SYSTEM DRILL_MVCL (* Drill System Model+View+Control+HMI with shared simulation clock *)
  (* Standard: 61499-1; Classification: Simulation; ApplicationDomain: Transfer Lines; Function: Drilling *)
  (* Version 0.2, 2007-07-07, JHC, Holobloc Inc, Added MODEL.CLOCK.CLK_DLY. *)
  (* Version 0.1, 2006-03-06, JHC, Holobloc Inc, Modified for new MACH_CTL. *)
  (* Version 0.0, 2004-09-26, JHC, Rockwell Automation, Derived from DRILL_MVL. *)
  DEVICE MODEL : FRAME_DEVICE(BOUNDS := [475,100,190,360])
    RESOURCE CLOCK : EMB_RES
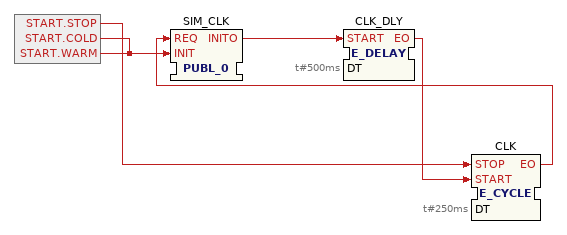
      FBS
        CLK : E_CYCLE(DT := t#250ms);
        SIM_CLK : PUBL_0;
        CLK_DLY : E_DELAY(DT := t#500ms); (* Wait for everything to initialize, then start simulation *)
      END_FBS
      EVENT_CONNECTIONS
        CLK.EO TO SIM_CLK.REQ;
        START.STOP TO CLK.STOP;
        START.COLD TO SIM_CLK.INIT;
        START.WARM TO SIM_CLK.INIT;
        SIM_CLK.INITO TO CLK_DLY.START;
        CLK_DLY.EO TO CLK.START;
      END_CONNECTIONS
    END_RESOURCE
    RESOURCE SUPPLY_MDL : EMB_RES
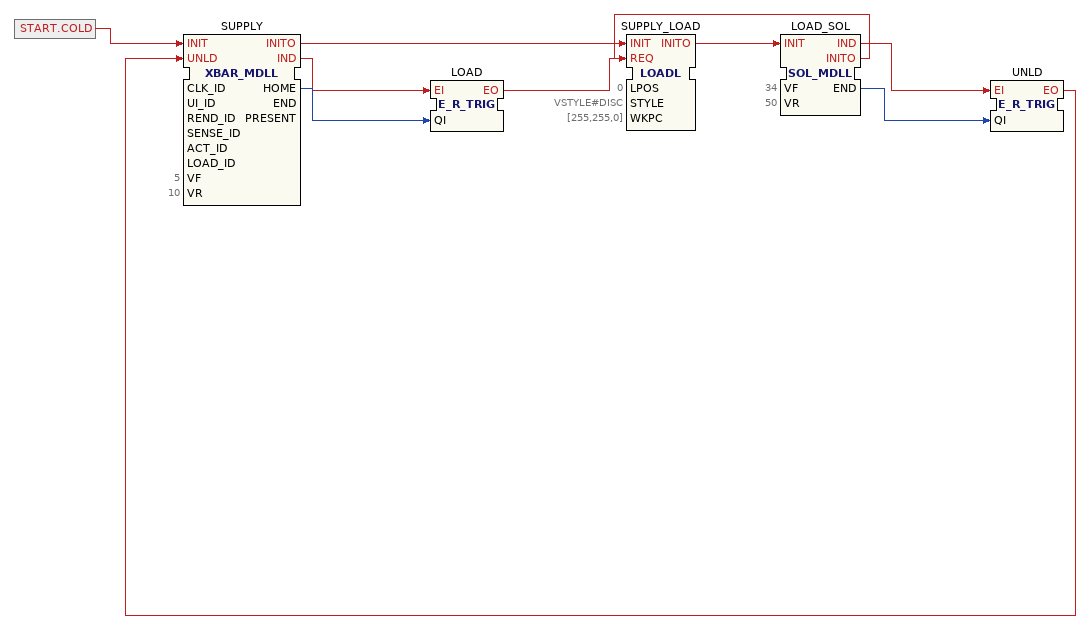
      FBS
        SUPPLY : XBAR_MDLL(VF := 5, VR := 10);
        LOAD_SOL : SOL_MDLL(VF := 34, VR := 50);
        UNLD : E_R_TRIG;
        LOAD : E_R_TRIG;
        SUPPLY_LOAD : LOADL(LPOS := 0, STYLE := VSTYLE#DISC, WKPC := [255,255,0]);
      END_FBS
      EVENT_CONNECTIONS
        START.COLD TO SUPPLY.INIT;
        LOAD_SOL.IND TO UNLD.EI;
        SUPPLY.IND TO LOAD.EI;
        UNLD.EO TO SUPPLY.UNLD;
        SUPPLY.INITO TO SUPPLY_LOAD.INIT;
        SUPPLY_LOAD.INITO TO LOAD_SOL.INIT;
        LOAD_SOL.INITO TO SUPPLY_LOAD.REQ;
        LOAD.EO TO SUPPLY_LOAD.REQ;
      END_CONNECTIONS
      DATA_CONNECTIONS
        LOAD_SOL.END TO UNLD.QI;
        SUPPLY.HOME TO LOAD.QI;
      END_CONNECTIONS
    END_RESOURCE
    RESOURCE SLIDE_MDL : EMB_RES
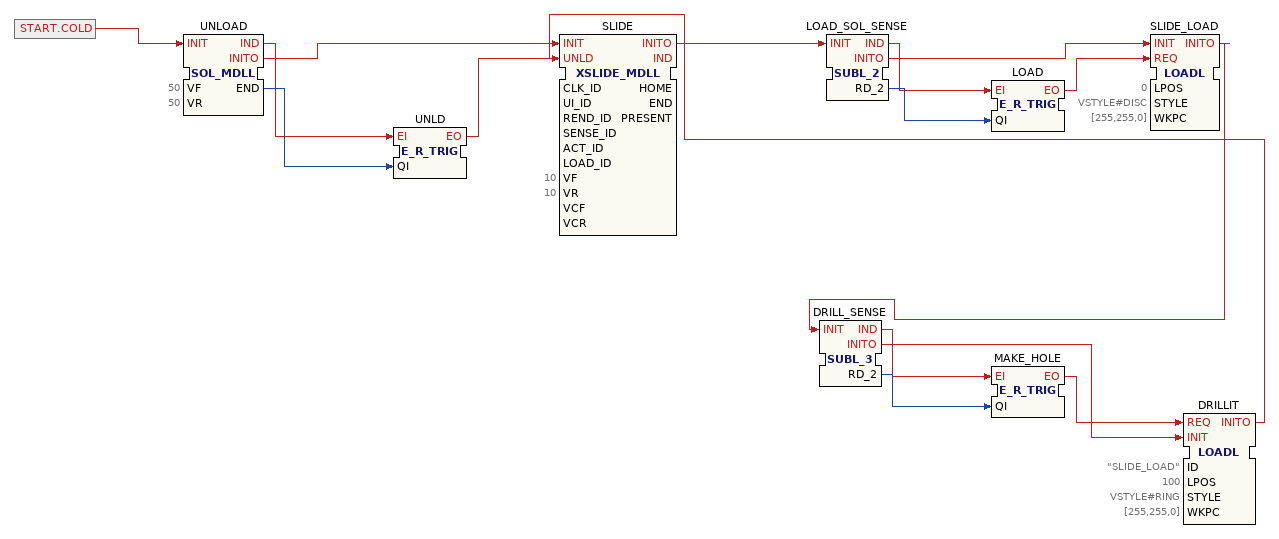
      FBS
        SLIDE : XSLIDE_MDLL(VF := 10, VR := 10);
        UNLOAD : SOL_MDLL(VF := 50, VR := 50);
        DRILL_SENSE : SUBL_3;
        MAKE_HOLE : E_R_TRIG;
        UNLD : E_R_TRIG;
        LOAD_SOL_SENSE : SUBL_2;
        LOAD : E_R_TRIG;
        SLIDE_LOAD : LOADL(LPOS := 0, STYLE := VSTYLE#DISC, WKPC := [255,255,0]);
        DRILLIT : LOADL(ID := "SLIDE_LOAD", LPOS := 100, STYLE := VSTYLE#RING, WKPC := [255,255,0]);
      END_FBS
      EVENT_CONNECTIONS
        DRILL_SENSE.IND TO MAKE_HOLE.EI;
        UNLOAD.IND TO UNLD.EI;
        UNLD.EO TO SLIDE.UNLD;
        LOAD_SOL_SENSE.IND TO LOAD.EI;
        START.COLD TO UNLOAD.INIT;
        UNLOAD.INITO TO SLIDE.INIT;
        SLIDE.INITO TO LOAD_SOL_SENSE.INIT;
        LOAD_SOL_SENSE.INITO TO SLIDE_LOAD.INIT;
        LOAD.EO TO SLIDE_LOAD.REQ;
        MAKE_HOLE.EO TO DRILLIT.REQ;
        DRILLIT.INITO TO SLIDE.UNLD;
        SLIDE_LOAD.INITO TO DRILL_SENSE.INIT;
        DRILL_SENSE.INITO TO DRILLIT.INIT;
      END_CONNECTIONS
      DATA_CONNECTIONS
        DRILL_SENSE.RD_2 TO MAKE_HOLE.QI;
        UNLOAD.END TO UNLD.QI;
        LOAD_SOL_SENSE.RD_2 TO LOAD.QI;
      END_CONNECTIONS
    END_RESOURCE
    RESOURCE DRILL_MDL : EMB_RES
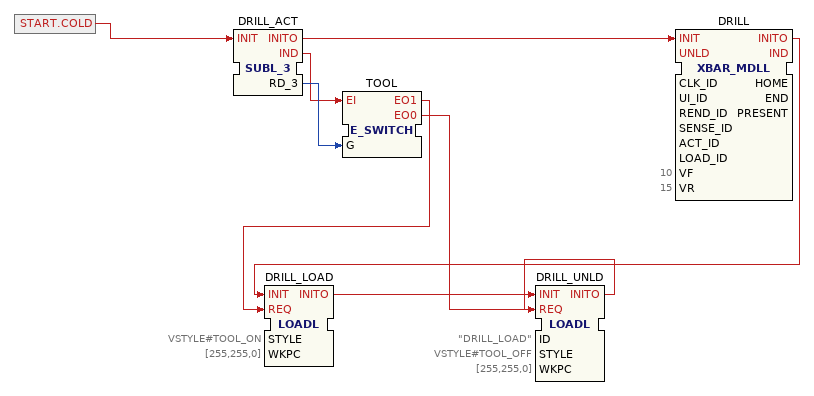
      FBS
        DRILL : XBAR_MDLL(VF := 10, VR := 15);
        DRILL_ACT : SUBL_3;
        TOOL : E_SWITCH;
        DRILL_LOAD : LOADL(STYLE := VSTYLE#TOOL_ON, WKPC := [255,255,0]);
        DRILL_UNLD : LOADL(ID := "DRILL_LOAD", STYLE := VSTYLE#TOOL_OFF, WKPC := [255,255,0]);
      END_FBS
      EVENT_CONNECTIONS
        START.COLD TO DRILL_ACT.INIT;
        DRILL_ACT.INITO TO DRILL.INIT;
        DRILL.INITO TO DRILL_LOAD.INIT;
        DRILL_LOAD.INITO TO DRILL_UNLD.INIT;
        DRILL_ACT.IND TO TOOL.EI;
        TOOL.EO1 TO DRILL_LOAD.REQ;
        TOOL.EO0 TO DRILL_UNLD.REQ;
        DRILL_UNLD.INITO TO DRILL_UNLD.REQ;
      END_CONNECTIONS
      DATA_CONNECTIONS
        DRILL_ACT.RD_3 TO TOOL.G;
      END_CONNECTIONS
    END_RESOURCE
    RESOURCE TAKEOFF_MDL : EMB_RES
      FBS
        UNLOAD_SENSE : SUBL_2;
        TAKEOFF : XBAR_MDLL(VF := 5, VR := 10);
        UNLD : E_R_TRIG;
        LOAD : E_R_TRIG;
        TAKEOFF_LOAD : LOADL(LPOS := 0, STYLE := VSTYLE#RING, WKPC := [255,255,0]);
      END_FBS
      EVENT_CONNECTIONS
        START.COLD TO UNLOAD_SENSE.INIT;
        UNLD.EO TO TAKEOFF.UNLD;
        TAKEOFF.IND TO UNLD.EI;
        TAKEOFF.INITO TO TAKEOFF.UNLD;
        UNLOAD_SENSE.IND TO LOAD.EI;
        UNLOAD_SENSE.INITO TO TAKEOFF_LOAD.INIT;
        TAKEOFF_LOAD.INITO TO TAKEOFF.INIT;
        LOAD.EO TO TAKEOFF_LOAD.REQ;
      END_CONNECTIONS
      DATA_CONNECTIONS
        TAKEOFF.END TO UNLD.QI;
        UNLOAD_SENSE.RD_2 TO LOAD.QI;
      END_CONNECTIONS
    END_RESOURCE
    RESOURCE INPUT_VIEW : VIEW_PANEL(DIA := 30, SIZE := [6,5], VERTICAL := 1)
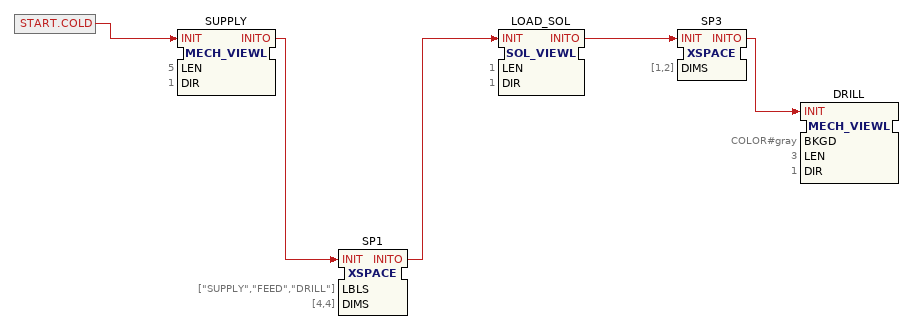
      FBS
        SUPPLY : MECH_VIEWL(LEN := 5, DIR := 1); (* Supply transfer mechanism *)
        SP1 : XSPACE(LBLS := ["SUPPLY","FEED","DRILL"], DIMS := [4,4]);
        LOAD_SOL : SOL_VIEWL(LEN := 1, DIR := 1); (* Loader mechanism *)
        SP3 : XSPACE(DIMS := [1,2]);
        DRILL : MECH_VIEWL(BKGD := COLOR#gray, LEN := 3, DIR := 1);
      END_FBS
      EVENT_CONNECTIONS
        START.COLD TO SUPPLY.INIT;
        SUPPLY.INITO TO SP1.INIT;
        SP1.INITO TO LOAD_SOL.INIT;
        LOAD_SOL.INITO TO SP3.INIT;
        SP3.INITO TO DRILL.INIT;
      END_CONNECTIONS
    END_RESOURCE
    RESOURCE OUTPUT_VIEW : VIEW_PANEL(DIA := 30, SIZE := [6,5])
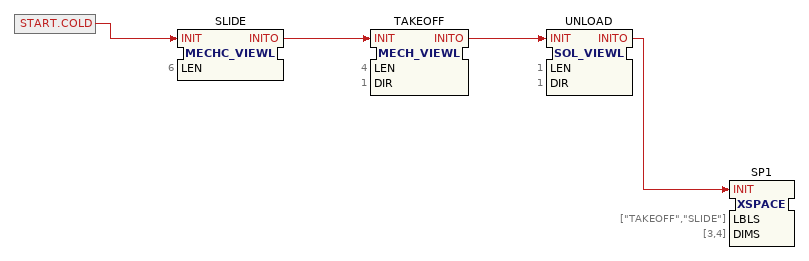
      FBS
        SLIDE : MECHC_VIEWL(LEN := 6);
        TAKEOFF : MECH_VIEWL(LEN := 4, DIR := 1); (* Takeoff Transfer *)
        UNLOAD : SOL_VIEWL(LEN := 1, DIR := 1); (* Unloader Mechanism *)
        SP1 : XSPACE(LBLS := ["TAKEOFF","SLIDE"], DIMS := [3,4]);
      END_FBS
      EVENT_CONNECTIONS
        START.COLD TO SLIDE.INIT;
        SLIDE.INITO TO TAKEOFF.INIT;
        TAKEOFF.INITO TO UNLOAD.INIT;
        UNLOAD.INITO TO SP1.INIT;
      END_CONNECTIONS
    END_RESOURCE
  END_DEVICE
  DEVICE CONTROL : FRAME_DEVICE(BOUNDS := [100,100,375,360], GRID := [6,2])
    RESOURCE SUPPLY_SENSORS : PANEL_RESOURCE
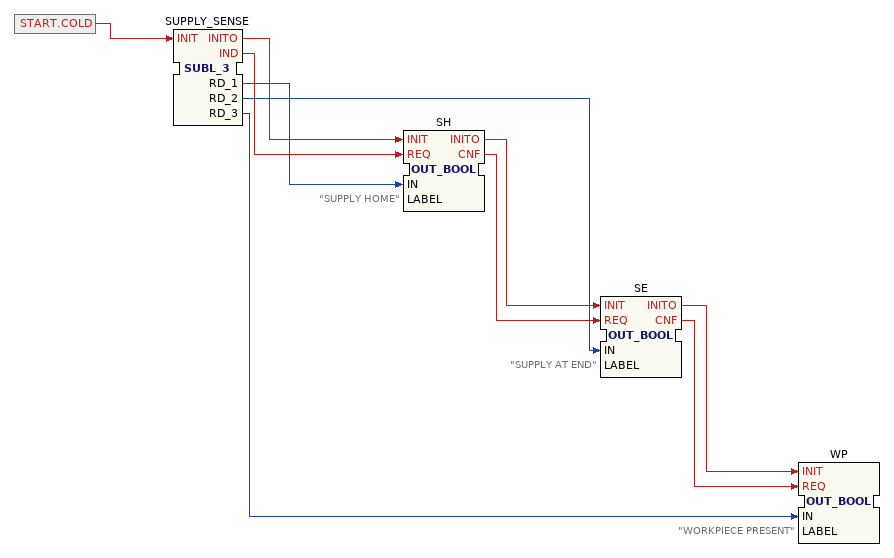
      FBS
        SUPPLY_SENSE : SUBL_3;
        SH : OUT_BOOL(LABEL := "SUPPLY HOME");
        SE : OUT_BOOL(LABEL := "SUPPLY AT END");
        WP : OUT_BOOL(LABEL := "WORKPIECE PRESENT");
      END_FBS
      EVENT_CONNECTIONS
        START.COLD TO SUPPLY_SENSE.INIT;
        SUPPLY_SENSE.INITO TO SH.INIT;
        SH.INITO TO SE.INIT;
        SE.INITO TO WP.INIT;
        SUPPLY_SENSE.IND TO SH.REQ;
        SH.CNF TO SE.REQ;
        SE.CNF TO WP.REQ;
      END_CONNECTIONS
      DATA_CONNECTIONS
        SUPPLY_SENSE.RD_1 TO SH.IN;
        SUPPLY_SENSE.RD_2 TO SE.IN;
        SUPPLY_SENSE.RD_3 TO WP.IN;
      END_CONNECTIONS
    END_RESOURCE
    RESOURCE SUPPLY_ACTUATORS : PANEL_RESOURCE(ROWS := 3)
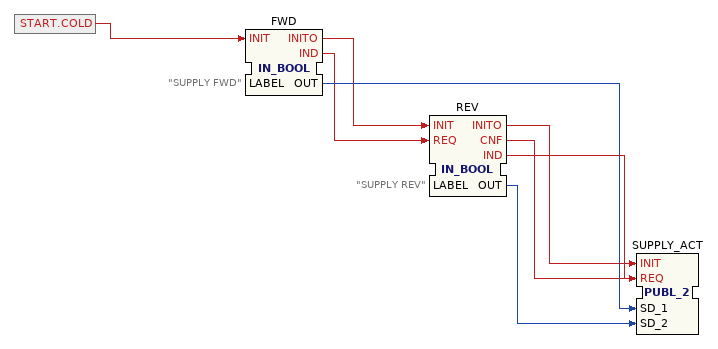
      FBS
        FWD : IN_BOOL(LABEL := "SUPPLY FWD");
        REV : IN_BOOL(LABEL := "SUPPLY REV");
        SUPPLY_ACT : PUBL_2;
      END_FBS
      EVENT_CONNECTIONS
        START.COLD TO FWD.INIT;
        FWD.INITO TO REV.INIT;
        REV.INITO TO SUPPLY_ACT.INIT;
        FWD.IND TO REV.REQ;
        REV.CNF TO SUPPLY_ACT.REQ;
        REV.IND TO SUPPLY_ACT.REQ;
      END_CONNECTIONS
      DATA_CONNECTIONS
        FWD.OUT TO SUPPLY_ACT.SD_1;
        REV.OUT TO SUPPLY_ACT.SD_2;
      END_CONNECTIONS
    END_RESOURCE
    RESOURCE LOAD_SENSORS : PANEL_RESOURCE
      FBS
        LOAD_SOL_SENSE : SUBL_2;
        HOME : OUT_BOOL(LABEL := "LOADER HOME");
        END : OUT_BOOL(LABEL := "LOADER AT END");
      END_FBS
      EVENT_CONNECTIONS
        START.COLD TO LOAD_SOL_SENSE.INIT;
        LOAD_SOL_SENSE.INITO TO HOME.INIT;
        HOME.INITO TO END.INIT;
        LOAD_SOL_SENSE.IND TO HOME.REQ;
        HOME.CNF TO END.REQ;
      END_CONNECTIONS
      DATA_CONNECTIONS
        LOAD_SOL_SENSE.RD_1 TO HOME.IN;
        LOAD_SOL_SENSE.RD_2 TO END.IN;
      END_CONNECTIONS
    END_RESOURCE
    RESOURCE LOAD_ACTUATORS : PANEL_RESOURCE(ROWS := 3)
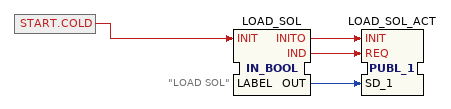
      FBS
        LOAD_SOL : IN_BOOL(LABEL := "LOAD SOL");
        LOAD_SOL_ACT : PUBL_1;
      END_FBS
      EVENT_CONNECTIONS
        START.COLD TO LOAD_SOL.INIT;
        LOAD_SOL.INITO TO LOAD_SOL_ACT.INIT;
        LOAD_SOL.IND TO LOAD_SOL_ACT.REQ;
      END_CONNECTIONS
      DATA_CONNECTIONS
        LOAD_SOL.OUT TO LOAD_SOL_ACT.SD_1;
      END_CONNECTIONS
    END_RESOURCE
    RESOURCE SLIDE_SENSORS : PANEL_RESOURCE
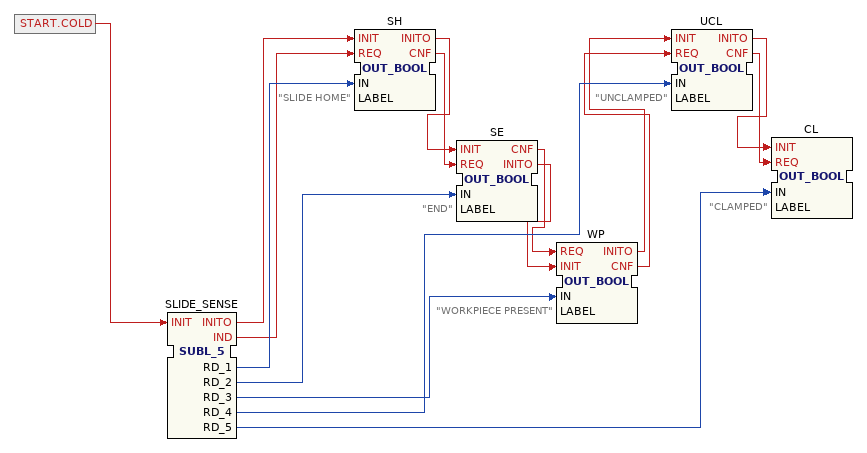
      FBS
        SLIDE_SENSE : SUBL_5;
        SH : OUT_BOOL(LABEL := "SLIDE HOME");
        SE : OUT_BOOL(LABEL := "END");
        UCL : OUT_BOOL(LABEL := "UNCLAMPED");
        CL : OUT_BOOL(LABEL := "CLAMPED");
        WP : OUT_BOOL(LABEL := "WORKPIECE PRESENT");
      END_FBS
      EVENT_CONNECTIONS
        START.COLD TO SLIDE_SENSE.INIT;
        SLIDE_SENSE.INITO TO SH.INIT;
        SH.INITO TO SE.INIT;
        UCL.INITO TO CL.INIT;
        SLIDE_SENSE.IND TO SH.REQ;
        SH.CNF TO SE.REQ;
        UCL.CNF TO CL.REQ;
        SE.CNF TO WP.REQ;
        SE.INITO TO WP.INIT;
        WP.INITO TO UCL.INIT;
        WP.CNF TO UCL.REQ;
      END_CONNECTIONS
      DATA_CONNECTIONS
        SLIDE_SENSE.RD_1 TO SH.IN;
        SLIDE_SENSE.RD_2 TO SE.IN;
        SLIDE_SENSE.RD_3 TO WP.IN;
        SLIDE_SENSE.RD_4 TO UCL.IN;
        SLIDE_SENSE.RD_5 TO CL.IN;
      END_CONNECTIONS
    END_RESOURCE
    RESOURCE SLIDE_ACTUATORS : PANEL_RESOURCE(ROWS := 3)
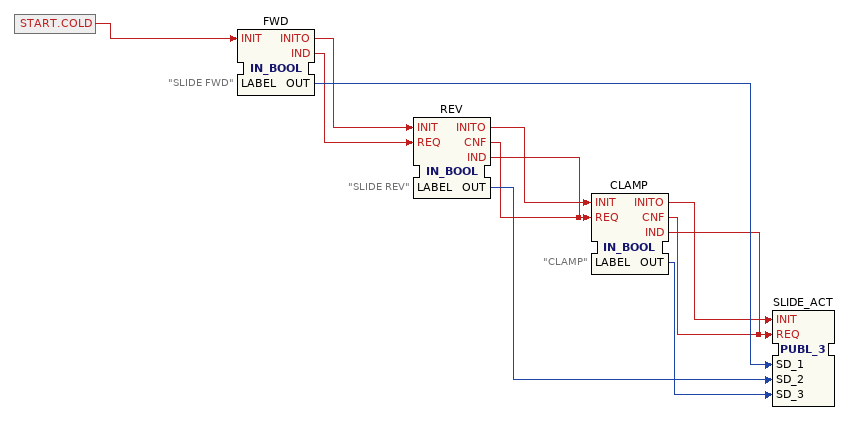
      FBS
        FWD : IN_BOOL(LABEL := "SLIDE FWD");
        REV : IN_BOOL(LABEL := "SLIDE REV");
        CLAMP : IN_BOOL(LABEL := "CLAMP");
        SLIDE_ACT : PUBL_3;
      END_FBS
      EVENT_CONNECTIONS
        START.COLD TO FWD.INIT;
        FWD.INITO TO REV.INIT;
        REV.INITO TO CLAMP.INIT;
        CLAMP.INITO TO SLIDE_ACT.INIT;
        FWD.IND TO REV.REQ;
        REV.CNF TO CLAMP.REQ;
        REV.IND TO CLAMP.REQ;
        CLAMP.CNF TO SLIDE_ACT.REQ;
        CLAMP.IND TO SLIDE_ACT.REQ;
      END_CONNECTIONS
      DATA_CONNECTIONS
        FWD.OUT TO SLIDE_ACT.SD_1;
        REV.OUT TO SLIDE_ACT.SD_2;
        CLAMP.OUT TO SLIDE_ACT.SD_3;
      END_CONNECTIONS
    END_RESOURCE
    RESOURCE DRILL_SENSORS : PANEL_RESOURCE
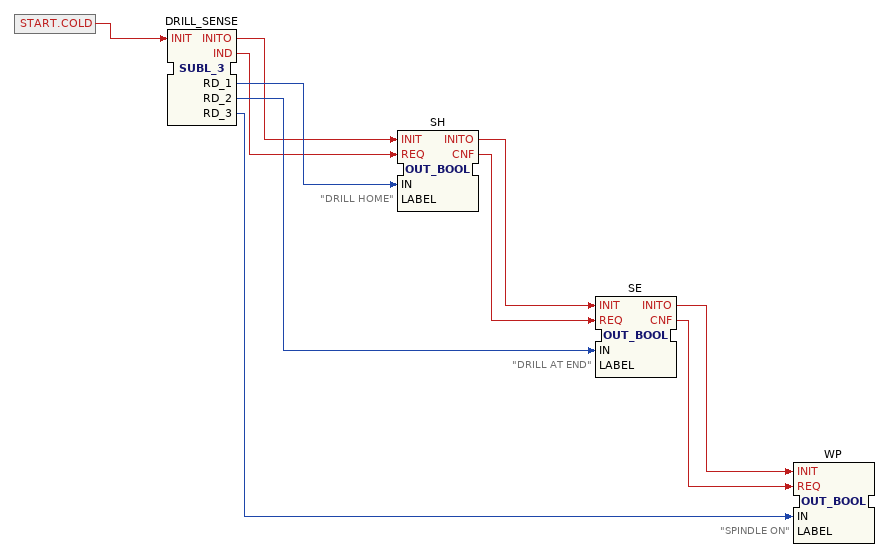
      FBS
        DRILL_SENSE : SUBL_3;
        SH : OUT_BOOL(LABEL := "DRILL HOME");
        SE : OUT_BOOL(LABEL := "DRILL AT END");
        WP : OUT_BOOL(LABEL := "SPINDLE ON");
      END_FBS
      EVENT_CONNECTIONS
        START.COLD TO DRILL_SENSE.INIT;
        DRILL_SENSE.INITO TO SH.INIT;
        SH.INITO TO SE.INIT;
        SE.INITO TO WP.INIT;
        DRILL_SENSE.IND TO SH.REQ;
        SH.CNF TO SE.REQ;
        SE.CNF TO WP.REQ;
      END_CONNECTIONS
      DATA_CONNECTIONS
        DRILL_SENSE.RD_1 TO SH.IN;
        DRILL_SENSE.RD_2 TO SE.IN;
        DRILL_SENSE.RD_3 TO WP.IN;
      END_CONNECTIONS
    END_RESOURCE
    RESOURCE DRILL_ACTUATORS : PANEL_RESOURCE(ROWS := 3)
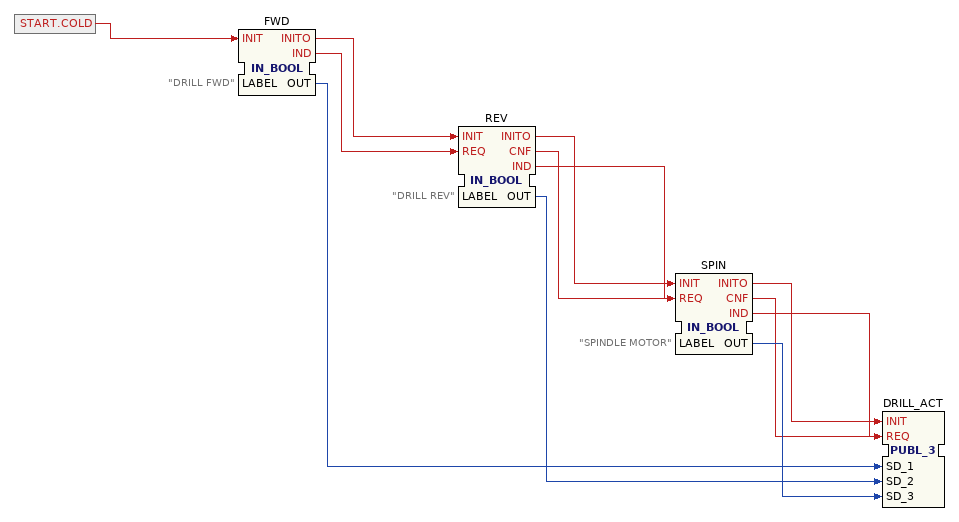
      FBS
        FWD : IN_BOOL(LABEL := "DRILL FWD");
        REV : IN_BOOL(LABEL := "DRILL REV");
        SPIN : IN_BOOL(LABEL := "SPINDLE MOTOR");
        DRILL_ACT : PUBL_3;
      END_FBS
      EVENT_CONNECTIONS
        START.COLD TO FWD.INIT;
        FWD.INITO TO REV.INIT;
        REV.INITO TO SPIN.INIT;
        SPIN.INITO TO DRILL_ACT.INIT;
        FWD.IND TO REV.REQ;
        REV.CNF TO SPIN.REQ;
        REV.IND TO SPIN.REQ;
        SPIN.CNF TO DRILL_ACT.REQ;
        SPIN.IND TO DRILL_ACT.REQ;
      END_CONNECTIONS
      DATA_CONNECTIONS
        FWD.OUT TO DRILL_ACT.SD_1;
        REV.OUT TO DRILL_ACT.SD_2;
        SPIN.OUT TO DRILL_ACT.SD_3;
      END_CONNECTIONS
    END_RESOURCE
    RESOURCE UNLOAD_SENSORS : PANEL_RESOURCE
      FBS
        UNLOAD_SENSE : SUBL_2;
        HOME : OUT_BOOL(LABEL := "UNLOADER HOME");
        END : OUT_BOOL(LABEL := "UNLOADER AT END");
      END_FBS
      EVENT_CONNECTIONS
        START.COLD TO UNLOAD_SENSE.INIT;
        UNLOAD_SENSE.INITO TO HOME.INIT;
        HOME.INITO TO END.INIT;
        UNLOAD_SENSE.IND TO HOME.REQ;
        HOME.CNF TO END.REQ;
      END_CONNECTIONS
      DATA_CONNECTIONS
        UNLOAD_SENSE.RD_1 TO HOME.IN;
        UNLOAD_SENSE.RD_2 TO END.IN;
      END_CONNECTIONS
    END_RESOURCE
    RESOURCE UNLOAD_ACTUATORS : PANEL_RESOURCE(ROWS := 3)
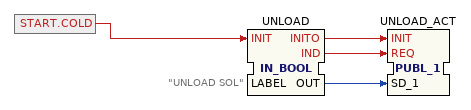
      FBS
        UNLOAD : IN_BOOL(LABEL := "UNLOAD SOL");
        UNLOAD_ACT : PUBL_1;
      END_FBS
      EVENT_CONNECTIONS
        START.COLD TO UNLOAD.INIT;
        UNLOAD.INITO TO UNLOAD_ACT.INIT;
        UNLOAD.IND TO UNLOAD_ACT.REQ;
      END_CONNECTIONS
      DATA_CONNECTIONS
        UNLOAD.OUT TO UNLOAD_ACT.SD_1;
      END_CONNECTIONS
    END_RESOURCE
    RESOURCE TAKEOFF_SENSORS : PANEL_RESOURCE
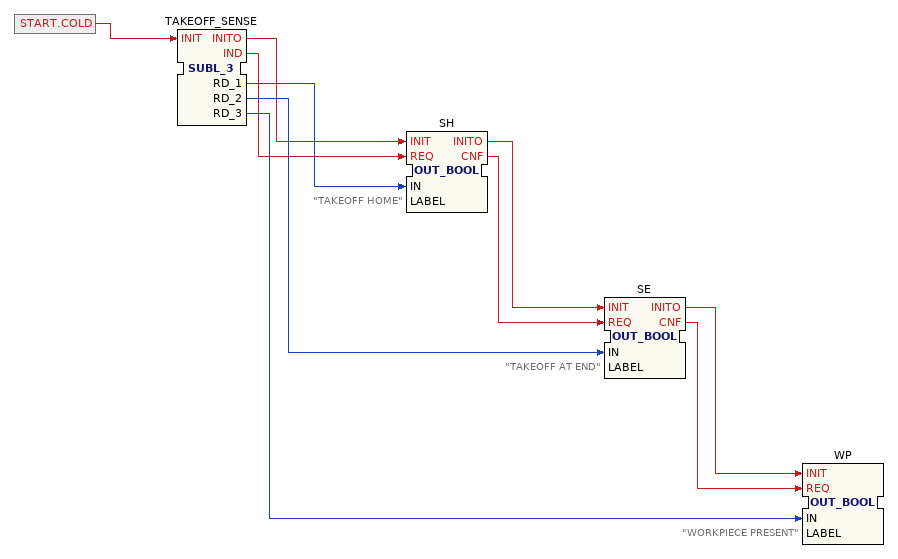
      FBS
        TAKEOFF_SENSE : SUBL_3;
        SH : OUT_BOOL(LABEL := "TAKEOFF HOME");
        SE : OUT_BOOL(LABEL := "TAKEOFF AT END");
        WP : OUT_BOOL(LABEL := "WORKPIECE PRESENT");
      END_FBS
      EVENT_CONNECTIONS
        START.COLD TO TAKEOFF_SENSE.INIT;
        TAKEOFF_SENSE.INITO TO SH.INIT;
        SH.INITO TO SE.INIT;
        SE.INITO TO WP.INIT;
        TAKEOFF_SENSE.IND TO SH.REQ;
        SH.CNF TO SE.REQ;
        SE.CNF TO WP.REQ;
      END_CONNECTIONS
      DATA_CONNECTIONS
        TAKEOFF_SENSE.RD_1 TO SH.IN;
        TAKEOFF_SENSE.RD_2 TO SE.IN;
        TAKEOFF_SENSE.RD_3 TO WP.IN;
      END_CONNECTIONS
    END_RESOURCE
    RESOURCE TAKEOFF_ACTUATORS : PANEL_RESOURCE(ROWS := 3)
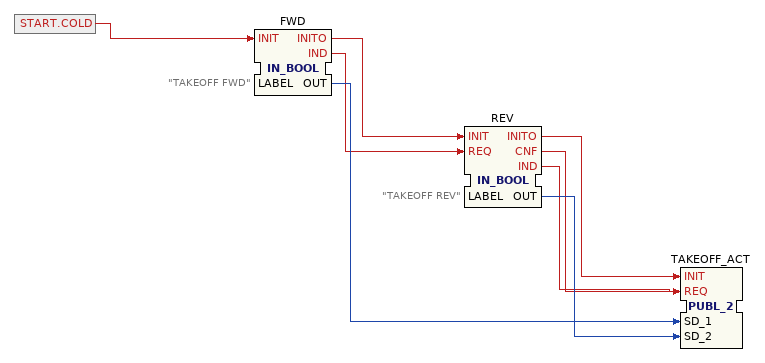
      FBS
        FWD : IN_BOOL(LABEL := "TAKEOFF FWD");
        REV : IN_BOOL(LABEL := "TAKEOFF REV");
        TAKEOFF_ACT : PUBL_2;
      END_FBS
      EVENT_CONNECTIONS
        START.COLD TO FWD.INIT;
        FWD.INITO TO REV.INIT;
        REV.INITO TO TAKEOFF_ACT.INIT;
        FWD.IND TO REV.REQ;
        REV.CNF TO TAKEOFF_ACT.REQ;
        REV.IND TO TAKEOFF_ACT.REQ;
      END_CONNECTIONS
      DATA_CONNECTIONS
        FWD.OUT TO TAKEOFF_ACT.SD_1;
        REV.OUT TO TAKEOFF_ACT.SD_2;
      END_CONNECTIONS
    END_RESOURCE
    RESOURCE SUPPLY : EMB_RES
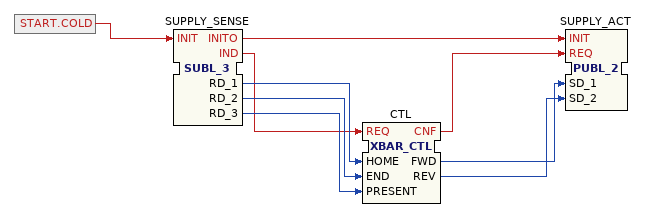
      FBS
        SUPPLY_SENSE : SUBL_3;
        CTL : XBAR_CTL;
        SUPPLY_ACT : PUBL_2;
      END_FBS
      EVENT_CONNECTIONS
        START.COLD TO SUPPLY_SENSE.INIT;
        SUPPLY_SENSE.INITO TO SUPPLY_ACT.INIT;
        SUPPLY_SENSE.IND TO CTL.REQ;
        CTL.CNF TO SUPPLY_ACT.REQ;
      END_CONNECTIONS
      DATA_CONNECTIONS
        SUPPLY_SENSE.RD_1 TO CTL.HOME;
        SUPPLY_SENSE.RD_2 TO CTL.END;
        SUPPLY_SENSE.RD_3 TO CTL.PRESENT;
        CTL.FWD TO SUPPLY_ACT.SD_1;
        CTL.REV TO SUPPLY_ACT.SD_2;
      END_CONNECTIONS
    END_RESOURCE
    RESOURCE LOAD : EMB_RES
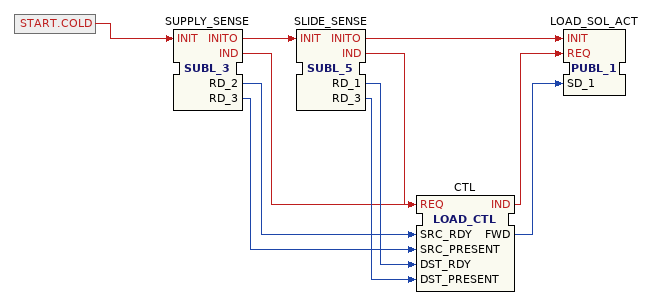
      FBS
        SUPPLY_SENSE : SUBL_3;
        SLIDE_SENSE : SUBL_5;
        CTL : LOAD_CTL;
        LOAD_SOL_ACT : PUBL_1;
      END_FBS
      EVENT_CONNECTIONS
        START.COLD TO SUPPLY_SENSE.INIT;
        SUPPLY_SENSE.INITO TO SLIDE_SENSE.INIT;
        SLIDE_SENSE.INITO TO LOAD_SOL_ACT.INIT;
        SUPPLY_SENSE.IND TO CTL.REQ;
        SLIDE_SENSE.IND TO CTL.REQ;
        CTL.IND TO LOAD_SOL_ACT.REQ;
      END_CONNECTIONS
      DATA_CONNECTIONS
        SUPPLY_SENSE.RD_2 TO CTL.SRC_RDY;
        SUPPLY_SENSE.RD_3 TO CTL.SRC_PRESENT;
        SLIDE_SENSE.RD_1 TO CTL.DST_RDY;
        CTL.FWD TO LOAD_SOL_ACT.SD_1;
        SLIDE_SENSE.RD_3 TO CTL.DST_PRESENT;
      END_CONNECTIONS
    END_RESOURCE
    RESOURCE SLIDE : EMB_RES
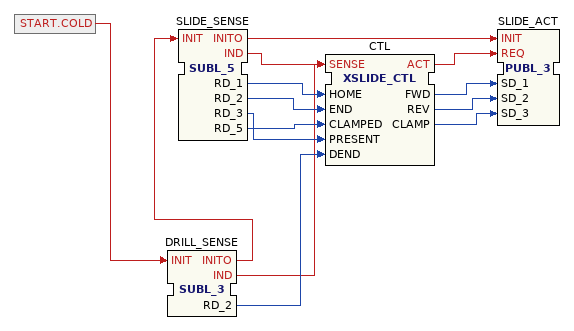
      FBS
        DRILL_SENSE : SUBL_3;
        SLIDE_SENSE : SUBL_5;
        CTL : XSLIDE_CTL;
        SLIDE_ACT : PUBL_3;
      END_FBS
      EVENT_CONNECTIONS
        START.COLD TO DRILL_SENSE.INIT;
        DRILL_SENSE.INITO TO SLIDE_SENSE.INIT;
        SLIDE_SENSE.INITO TO SLIDE_ACT.INIT;
        SLIDE_SENSE.IND TO CTL.SENSE;
        DRILL_SENSE.IND TO CTL.SENSE;
        CTL.ACT TO SLIDE_ACT.REQ;
      END_CONNECTIONS
      DATA_CONNECTIONS
        SLIDE_SENSE.RD_1 TO CTL.HOME;
        SLIDE_SENSE.RD_2 TO CTL.END;
        DRILL_SENSE.RD_2 TO CTL.DEND;
        CTL.FWD TO SLIDE_ACT.SD_1;
        CTL.REV TO SLIDE_ACT.SD_2;
        CTL.CLAMP TO SLIDE_ACT.SD_3;
        SLIDE_SENSE.RD_3 TO CTL.PRESENT;
        SLIDE_SENSE.RD_5 TO CTL.CLAMPED;
      END_CONNECTIONS
    END_RESOURCE
    RESOURCE DRILL : EMB_RES
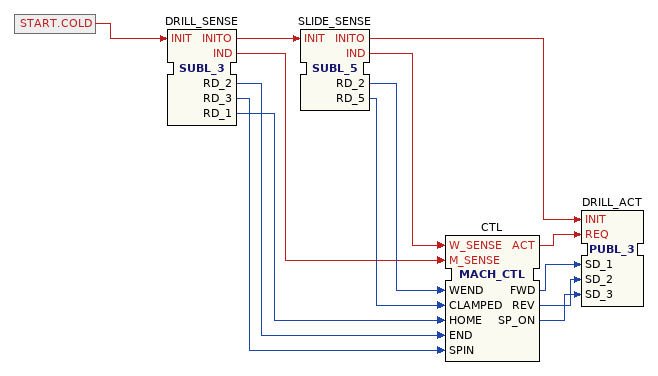
      FBS
        DRILL_SENSE : SUBL_3;
        SLIDE_SENSE : SUBL_5;
        CTL : MACH_CTL;
        DRILL_ACT : PUBL_3;
      END_FBS
      EVENT_CONNECTIONS
        START.COLD TO DRILL_SENSE.INIT;
        DRILL_SENSE.INITO TO SLIDE_SENSE.INIT;
        SLIDE_SENSE.INITO TO DRILL_ACT.INIT;
        CTL.ACT TO DRILL_ACT.REQ;
        DRILL_SENSE.IND TO CTL.M_SENSE;
        SLIDE_SENSE.IND TO CTL.W_SENSE;
      END_CONNECTIONS
      DATA_CONNECTIONS
        SLIDE_SENSE.RD_2 TO CTL.WEND;
        DRILL_SENSE.RD_2 TO CTL.END;
        DRILL_SENSE.RD_3 TO CTL.SPIN;
        CTL.FWD TO DRILL_ACT.SD_1;
        CTL.REV TO DRILL_ACT.SD_2;
        CTL.SP_ON TO DRILL_ACT.SD_3;
        SLIDE_SENSE.RD_5 TO CTL.CLAMPED;
        DRILL_SENSE.RD_1 TO CTL.HOME;
      END_CONNECTIONS
    END_RESOURCE
    RESOURCE UNLOAD : EMB_RES
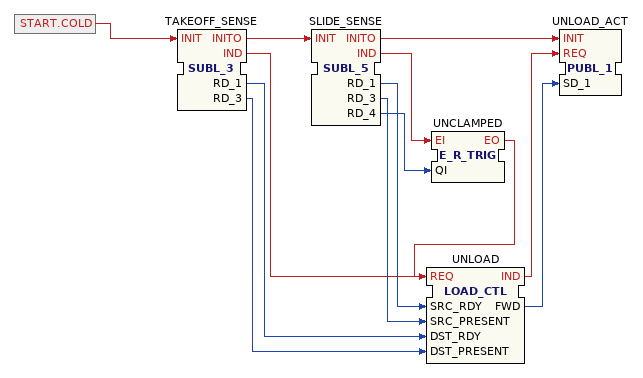
      FBS
        SLIDE_SENSE : SUBL_5;
        TAKEOFF_SENSE : SUBL_3;
        UNLOAD : LOAD_CTL;
        UNLOAD_ACT : PUBL_1;
        UNCLAMPED : E_R_TRIG;
      END_FBS
      EVENT_CONNECTIONS
        START.COLD TO TAKEOFF_SENSE.INIT;
        TAKEOFF_SENSE.INITO TO SLIDE_SENSE.INIT;
        SLIDE_SENSE.INITO TO UNLOAD_ACT.INIT;
        TAKEOFF_SENSE.IND TO UNLOAD.REQ;
        UNLOAD.IND TO UNLOAD_ACT.REQ;
        SLIDE_SENSE.IND TO UNCLAMPED.EI;
        UNCLAMPED.EO TO UNLOAD.REQ;
      END_CONNECTIONS
      DATA_CONNECTIONS
        TAKEOFF_SENSE.RD_1 TO UNLOAD.DST_RDY;
        TAKEOFF_SENSE.RD_3 TO UNLOAD.DST_PRESENT;
        SLIDE_SENSE.RD_1 TO UNLOAD.SRC_RDY;
        UNLOAD.FWD TO UNLOAD_ACT.SD_1;
        SLIDE_SENSE.RD_3 TO UNLOAD.SRC_PRESENT;
        SLIDE_SENSE.RD_4 TO UNCLAMPED.QI;
      END_CONNECTIONS
    END_RESOURCE
    RESOURCE TAKEOFF : EMB_RES
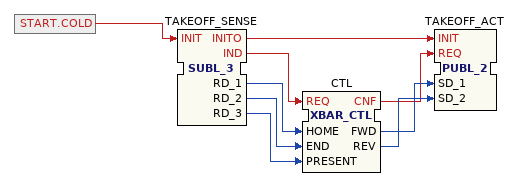
      FBS
        TAKEOFF_SENSE : SUBL_3;
        CTL : XBAR_CTL;
        TAKEOFF_ACT : PUBL_2;
      END_FBS
      EVENT_CONNECTIONS
        START.COLD TO TAKEOFF_SENSE.INIT;
        TAKEOFF_SENSE.INITO TO TAKEOFF_ACT.INIT;
        TAKEOFF_SENSE.IND TO CTL.REQ;
        CTL.CNF TO TAKEOFF_ACT.REQ;
      END_CONNECTIONS
      DATA_CONNECTIONS
        TAKEOFF_SENSE.RD_1 TO CTL.HOME;
        TAKEOFF_SENSE.RD_2 TO CTL.END;
        TAKEOFF_SENSE.RD_3 TO CTL.PRESENT;
        CTL.FWD TO TAKEOFF_ACT.SD_1;
        CTL.REV TO TAKEOFF_ACT.SD_2;
      END_CONNECTIONS
    END_RESOURCE
  END_DEVICE
END_SYSTEM
